TYPE Router :
STRUCT
		MesWatchdog	        : BOOL ; 	(* Watchdog*)
		
		MesAlarmCode		: WORD ;	(* (NA) Internal Akuo AlarmCode		*)
		MesWarningCode		: WORD ; 	(* (NA) Internal Akuo WarningCode   *)
		MesEventCode		: WORD ; 	(* (NA) Internal Akuo EventCode	    *)
		
END_STRUCT
END_TYPE

(* stored: Version 1.1.0.1, ProductVersion 3.1.4024.6
   DUT Router: Id {dbad6274-51a4-41cc-8bf7-03e6125eb91c} *)
